FUNCTION IsValidInputPort : BOOL
VAR_INPUT
	InputPort : I_InputPort;
END_VAR

IsValidInputPort := InputPort <> 0;

END_FUNCTION

(* stored: Version 1.1.0.1, ProductVersion 3.1.4024.12
   POU IsValidInputPort: Id {1ee37e81-2a18-025e-2a8e-aaa7ade41a36}, SpecialFunc None *)
